// Mitsubishi GX Works2 project: Auto Batch and Spray   PLC: FX1N/FX1NC

// global labels: Global1
VAR_GLOBAL
  senMolasses AT X000 : BOOL;
  senDischargeMol AT X001 : BOOL;
  senCocoOil AT X002 : BOOL;
  senDischargeCoco AT X003 : BOOL;
  rStartMolasses AT Y000 : BOOL;
  rDischargeMolasses AT Y001 : BOOL;
  rStopMolasses AT Y002 : BOOL;
  rStartCocoOil AT Y003 : BOOL;
  rDischargeCocoOil AT Y004 : BOOL;
  rStopCocoOil AT Y005 : BOOL;
  inStart AT X004 : BOOL;
  inStop AT X005 : BOOL;
  inEnMolasses AT X006 : BOOL;
  inEnCocoOil AT X007 : BOOL;
  RunAutoFlag : BOOL;
  RunAutoMolassesStatus : INT;
  RunAutoCocoOilStatus : INT;
END_VAR
VAR_GLOBAL CONSTANT
  SprayTimeAfterDischargeMol : TIME := T#60s;
  SprayTimeAfterDischargeCoco : TIME := T#60s;
END_VAR

// task Task_01 (event TRUE, interval 0, priority 31): POU_01

PROGRAM POU_01
VAR
  OutputRStartMolasses : RunOutput;
  OutputRStopMolasses : RunOutput;
  OutputRDischargeMolasses : RunOutput;
  OutputRStartCocoOil : RunOutput;
  OutputRStopCocoOil : RunOutput;
  OutputRDischargeCocoOil : RunOutput;
END_VAR
(* Start Run Auto *)
IF	inStart= TRUE THEN
	RunAutoFlag:= TRUE;
	RunAutoMolassesStatus:=1;
  	RunAutoCocoOilStatus:= 1;
END_IF;

(* Stop Alll *)
IF inStop= TRUE THEN
	runAutoFlag := FALSE;
	RunAutoCocoOilStatus:=0;
	RunAutoMolassesStatus:=0;
	rStartMolasses:=FALSE;
	rStopMolasses:=FALSE;
	rDischargeMolasses:=FALSE;
	rStartCocoOil:=FALSE;
	rStopCocoOil:=FALSE;
	rDischargeCocoOil:=FALSE;
END_IF;

OutputRStartMolasses(input:= rStartMolasses ,output:= rStartMolasses);
OutputRStopMolasses(input:= rStopMolasses ,output:= rStopMolasses);
OutputRDischargeMolasses(input:= rDischargeMolasses ,output:= rDischargeMolasses);
OutputRStartCocoOil(input:= rStartCocoOil ,output:= rStartCocoOil);
OutputRStopCocoOil(input:= rStopCocoOil ,output:= rStopCocoOil);
OutputRDischargeCocoOil(input:= rDischargeCocoOil ,output:= rDischargeCocoOil);
END_PROGRAM

FUNCTION_BLOCK RunOutput
VAR_INPUT
  input : BOOL;
END_VAR
VAR_OUTPUT
  output : BOOL;
END_VAR
(* structured ladder/FBD written out as ST: instructions are called as NAME(EN, inputs, outputs); _pN, _eN, _tN stand for wires *)
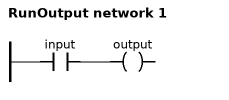
(* network 1 *)
output := input;
END_FUNCTION_BLOCK
